// TIA Portal V18 export
// export: Created 2025-12-01T17:51:19.9261782Z, ExportSetting None, DisplayName Totally Integrated Automation Portal, DisplayVersion V18 Update 5, DisplayName TIA Portal Openness, DisplayVersion V18 Update 5, DisplayName TIA Portal Teamcenter Gateway, DisplayVersion V18, DisplayName TIA Portal Version Control Interface, DisplayVersion V18, DisplayName STEP 7 Professional, DisplayVersion V18 Update 5, DisplayName STEP 7 Safety, DisplayVersion V18, DisplayName WinCC Professional, DisplayVersion V18 Update 5
FUNCTION_BLOCK "MotorContro"   // FB3100, LAD
{ S7_Optimized_Access := 'TRUE' }
// stored: AutoNumber false, MemoryReserve 100, SetENOAutomatically false
   VAR_INPUT
      iAlwaysTrue : Bool;
      iSysRun : Bool;
      iReset : Bool;
      iAuto : Bool;
      iManual : Bool;
      i_ParySensor : Bool;
      i_Alarm : Bool;
      iType : Int;
      i_RunInTimeDelay : Time;
      i_RunOutTimeDelay : Time;
      i_Interlock : Bool;
   END_VAR
   VAR_IN_OUT
      Control : "Motor_Control";
   END_VAR
   VAR
      TON : Array[0..5] of TON_TIME;
      Zero { S7_SetPoint := 'True'} : Array[0..15] of Bool;
   END_VAR
   VAR_TEMP   // added for the SCL form of the ladder/FBD networks
      _w1 : Bool;
   END_VAR
BEGIN

REGION Network 1: Reset
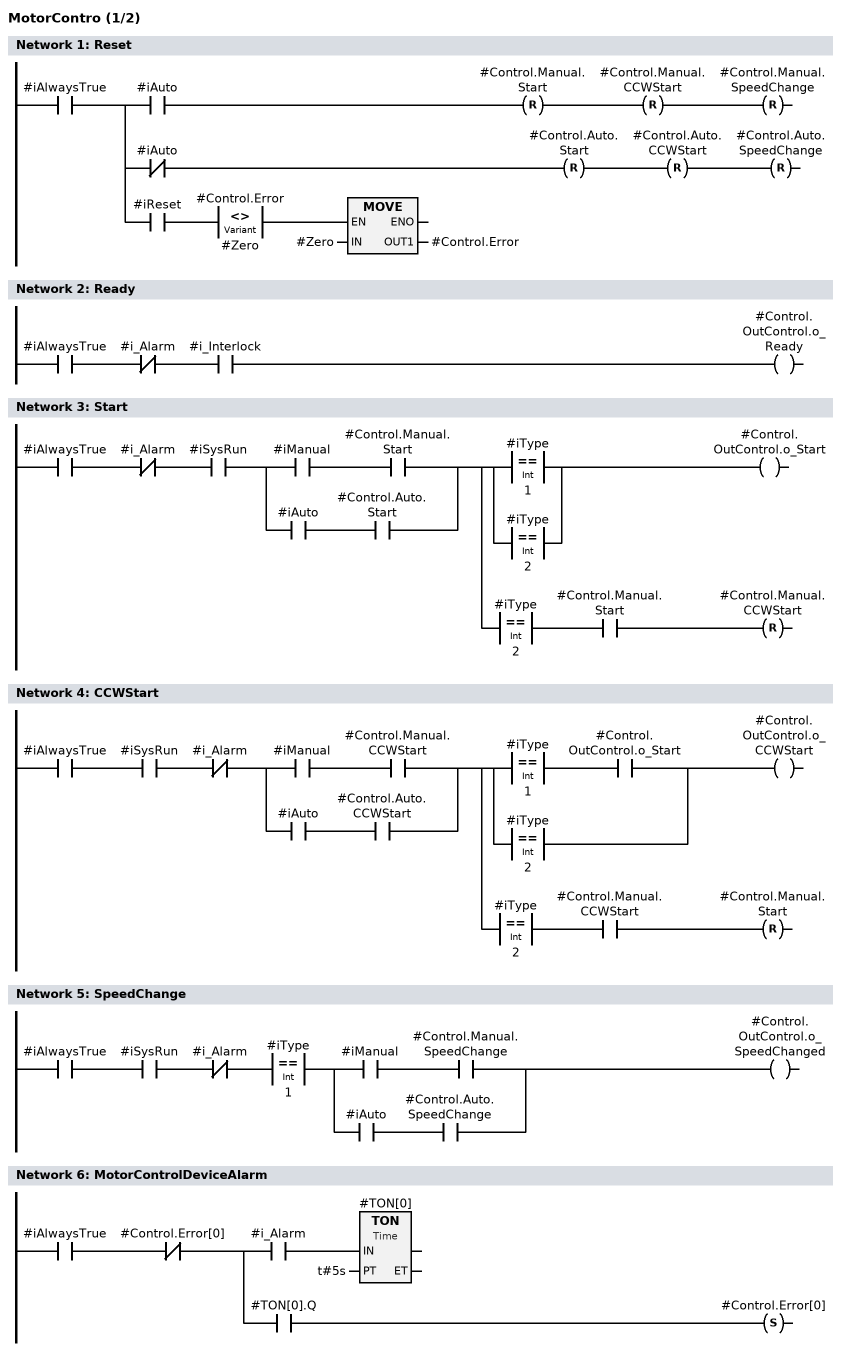
   RUNG wire#powerrail
      Contact( #iAlwaysTrue )
      wire#w1
      Contact( #iAuto )
      R_Coil( #Control.Manual.Start )
      R_Coil( #Control.Manual.CCWStart )
      R_Coil( #Control.Manual.SpeedChange )
   END_RUNG
   RUNG wire#w1
      I_Contact( #iAuto )
      R_Coil( #Control.Auto.Start )
      R_Coil( #Control.Auto.CCWStart )
      R_Coil( #Control.Auto.SpeedChange )
   END_RUNG
   RUNG wire#w1
      Contact( #iReset )
      { S7_Templates := "SrcType := Variant" } NE_Contact(in1 := #Control.Error, in2 := #Zero)
      Move(in := #Zero, out1 => #Control.Error)
   END_RUNG
   // the same network as SCL:
   IF #iAlwaysTrue AND #iAuto THEN
       #Control.Manual.Start := FALSE;
       #Control.Manual.CCWStart := FALSE;
       #Control.Manual.SpeedChange := FALSE;
   END_IF;
   IF #iAlwaysTrue AND NOT #iAuto THEN
       #Control.Auto.Start := FALSE;
       #Control.Auto.CCWStart := FALSE;
       #Control.Auto.SpeedChange := FALSE;
   END_IF;
   IF #iAlwaysTrue AND #iReset AND (#Control.Error <> #Zero) THEN #Control.Error := #Zero; END_IF;
END_REGION

REGION Network 2: Ready
   RUNG wire#powerrail
      Contact( #iAlwaysTrue )
      I_Contact( #i_Alarm )
      Contact( #i_Interlock )
      Coil( #Control.OutControl.o_Ready )
   END_RUNG
   // the same network as SCL:
   #Control.OutControl.o_Ready := #iAlwaysTrue AND NOT #i_Alarm AND #i_Interlock;
END_REGION

REGION Network 3: Start
   RUNG wire#powerrail
      Contact( #iAlwaysTrue )
      I_Contact( #i_Alarm )
      Contact( #iSysRun )
      wire#w1
      Contact( #iManual )
      Contact( #Control.Manual.Start )
      wire#w2
      { S7_Templates := "SrcType := Int" } EQ_Contact(in1 := #iType, in2 := 1)
      wire#w3
      Coil( #Control.OutControl.o_Start )
   END_RUNG
   RUNG wire#w1
      Contact( #iAuto )
      Contact( #Control.Auto.Start )
   END_RUNG wire#w2
   RUNG wire#w2
      { S7_Templates := "SrcType := Int" } EQ_Contact(in1 := #iType, in2 := 2)
   END_RUNG wire#w3
   RUNG wire#w2
      { S7_Templates := "SrcType := Int" } EQ_Contact(in1 := #iType, in2 := 2)
      Contact( #Control.Manual.Start )
      R_Coil( #Control.Manual.CCWStart )
   END_RUNG
   // the same network as SCL:
   #_w1 := #iAlwaysTrue AND NOT #i_Alarm AND #iSysRun AND ((#iManual AND #Control.Manual.Start) OR (#iAuto AND #Control.Auto.Start));
   #Control.OutControl.o_Start := #_w1 AND ((#iType = 1) OR (#iType = 2));
   IF #_w1 AND (#iType = 2) AND #Control.Manual.Start THEN #Control.Manual.CCWStart := FALSE; END_IF;
END_REGION

REGION Network 4: CCWStart
   RUNG wire#powerrail
      Contact( #iAlwaysTrue )
      Contact( #iSysRun )
      I_Contact( #i_Alarm )
      wire#w1
      Contact( #iManual )
      Contact( #Control.Manual.CCWStart )
      wire#w2
      { S7_Templates := "SrcType := Int" } EQ_Contact(in1 := #iType, in2 := 1)
      Contact( #Control.OutControl.o_Start )
      wire#w3
      Coil( #Control.OutControl.o_CCWStart )
   END_RUNG
   RUNG wire#w1
      Contact( #iAuto )
      Contact( #Control.Auto.CCWStart )
   END_RUNG wire#w2
   RUNG wire#w2
      { S7_Templates := "SrcType := Int" } EQ_Contact(in1 := #iType, in2 := 2)
   END_RUNG wire#w3
   RUNG wire#w2
      { S7_Templates := "SrcType := Int" } EQ_Contact(in1 := #iType, in2 := 2)
      Contact( #Control.Manual.CCWStart )
      R_Coil( #Control.Manual.Start )
   END_RUNG
   // the same network as SCL:
   #_w1 := #iAlwaysTrue AND #iSysRun AND NOT #i_Alarm AND ((#iManual AND #Control.Manual.CCWStart) OR (#iAuto AND #Control.Auto.CCWStart));
   #Control.OutControl.o_CCWStart := #_w1 AND (((#iType = 1) AND #Control.OutControl.o_Start) OR (#iType = 2));
   IF #_w1 AND (#iType = 2) AND #Control.Manual.CCWStart THEN #Control.Manual.Start := FALSE; END_IF;
END_REGION

REGION Network 5: SpeedChange
   RUNG wire#powerrail
      Contact( #iAlwaysTrue )
      Contact( #iSysRun )
      I_Contact( #i_Alarm )
      { S7_Templates := "SrcType := Int" } EQ_Contact(in1 := #iType, in2 := 1)
      wire#w1
      Contact( #iManual )
      Contact( #Control.Manual.SpeedChange )
      wire#w2
      Coil( #Control.OutControl.o_SpeedChanged )
   END_RUNG
   RUNG wire#w1
      Contact( #iAuto )
      Contact( #Control.Auto.SpeedChange )
   END_RUNG wire#w2
   // the same network as SCL:
   #Control.OutControl.o_SpeedChanged := #iAlwaysTrue AND #iSysRun AND NOT #i_Alarm AND (#iType = 1) AND ((#iManual AND #Control.Manual.SpeedChange) OR (#iAuto AND #Control.Auto.SpeedChange));
END_REGION

REGION Network 6: MotorControlDeviceAlarm
   RUNG wire#powerrail
      Contact( #iAlwaysTrue )
      I_Contact( #Control.Error[0] )
      wire#w1
      Contact( #i_Alarm )
      { S7_Templates := "time_type := Time" } #TON[0].TON(pt := t#5s, et =>)
   END_RUNG
   RUNG wire#w1
      Contact( #TON[0].Q )
      S_Coil( #Control.Error[0] )
   END_RUNG
   // the same network as SCL:
   #_w1 := #iAlwaysTrue AND NOT #Control.Error[0];
   #TON[0].TON(IN := #_w1 AND #i_Alarm, PT := t#5s);
   IF #_w1 AND #TON[0].Q THEN #Control.Error[0] := TRUE; END_IF;
END_REGION

REGION Network 7: PalletRunInTimeOut
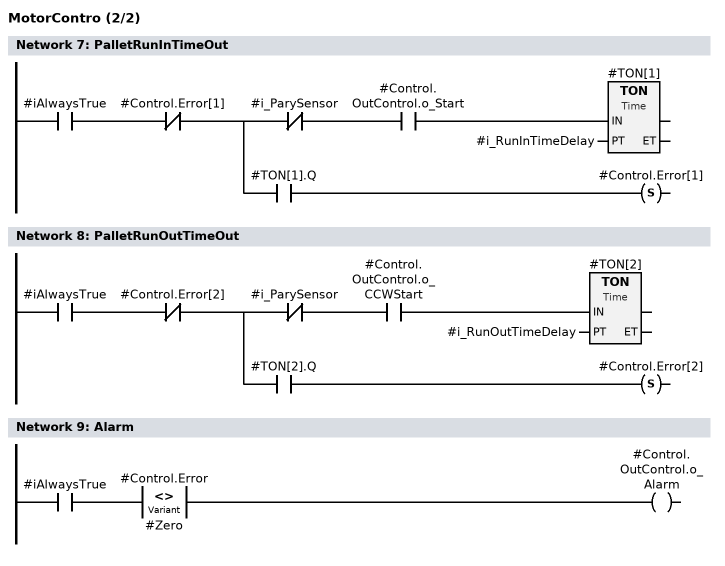
   RUNG wire#powerrail
      Contact( #iAlwaysTrue )
      I_Contact( #Control.Error[1] )
      wire#w1
      I_Contact( #i_ParySensor )
      Contact( #Control.OutControl.o_Start )
      { S7_Templates := "time_type := Time" } #TON[1].TON(pt := #i_RunInTimeDelay, et =>)
   END_RUNG
   RUNG wire#w1
      Contact( #TON[1].Q )
      S_Coil( #Control.Error[1] )
   END_RUNG
   // the same network as SCL:
   #_w1 := #iAlwaysTrue AND NOT #Control.Error[1];
   #TON[1].TON(IN := #_w1 AND NOT #i_ParySensor AND #Control.OutControl.o_Start, PT := #i_RunInTimeDelay);
   IF #_w1 AND #TON[1].Q THEN #Control.Error[1] := TRUE; END_IF;
END_REGION

REGION Network 8: PalletRunOutTimeOut
   RUNG wire#powerrail
      Contact( #iAlwaysTrue )
      I_Contact( #Control.Error[2] )
      wire#w1
      I_Contact( #i_ParySensor )
      Contact( #Control.OutControl.o_CCWStart )
      { S7_Templates := "time_type := Time" } #TON[2].TON(pt := #i_RunOutTimeDelay, et =>)
   END_RUNG
   RUNG wire#w1
      Contact( #TON[2].Q )
      S_Coil( #Control.Error[2] )
   END_RUNG
   // the same network as SCL:
   #_w1 := #iAlwaysTrue AND NOT #Control.Error[2];
   #TON[2].TON(IN := #_w1 AND NOT #i_ParySensor AND #Control.OutControl.o_CCWStart, PT := #i_RunOutTimeDelay);
   IF #_w1 AND #TON[2].Q THEN #Control.Error[2] := TRUE; END_IF;
END_REGION

REGION Network 9: Alarm
   RUNG wire#powerrail
      Contact( #iAlwaysTrue )
      { S7_Templates := "SrcType := Variant" } NE_Contact(in1 := #Control.Error, in2 := #Zero)
      Coil( #Control.OutControl.o_Alarm )
   END_RUNG
   // the same network as SCL:
   #Control.OutControl.o_Alarm := #iAlwaysTrue AND (#Control.Error <> #Zero);
END_REGION
END_FUNCTION_BLOCK
